(* Test enum. *)
TYPE E_TestMode : (
    Off := 0,
    On  := 1  (* Active state *)
);
END_TYPE

(* stored: Version 1.1.0.1
   DUT E_TestMode: Id {55555555-5555-5555-5555-555555555501} *)
